FUNCTION_BLOCK FB_TouchProbe
VAR_INPUT
	AxisIdx	:INT;
END_VAR
VAR_OUTPUT
END_VAR
VAR
END_VAR

AxisTouchProbe[AxisIdx].Execute := TRUE;

END_FUNCTION_BLOCK

(* stored: Version 1.1.0.1, ProductVersion 3.1.4024.9
   POU FB_TouchProbe: Id {1eb36dc9-79a4-42ba-b573-1d044a7b5f9d}, SpecialFunc None *)
